(* Schneider Machine Expert - Basic project MEB, file version 2.7.0.0 *)
(* ProjectInformations: Name=Novo projeto *)

HARDWARE
  Cpu 0: TM221CE24R
  EthernetConfiguration: NetworkName=M221, IpAllocationMode=FixedAddress, IpAddress=0.0.0.0, SubnetMask=0.0.0.0
  SerialLineConfiguration: Baud=Baud19200, Parity=ParityEven, DataBits=DataBits8, StopBits=StopBits1, PhysicalMedium=PhysicalMediumRs485, TransmissionMode=TransmissionModeModbusRtu, SlaveId=1, Addressing=SlaveAddressing
  MastTask: UsePeriodScanMode=false, PeriodScan=100
  FastTask: Period=255
  CpuBehavior: StartingMode=StartAsPreviousState, AutoSaveRamOnEeprom=true, WatchdogPeriod=250

SYMBOLS  (address, symbol, comment, settings)
  %M0       AUX_PAI_EMER
  %M1       AUX_PAI_LOCA
  %M2       AUX_PAI_REMO
  %M3       CMD_PAI_MOT1_LIGA
  %M4       CMD_PAI_MOT1_DESL
  %M5       CMD_PAI_MOT2_LIGA
  %M6       CMD_PAI_MOT2_DESL
  %M50      HAB_MOT1
  %M51      HAB_MOT2
  %M100     CMD_IHM_INICIO
  %M101     CMD_IHM_FIM
  %I0.0     PAI_EMER
  %I0.1     PAI_LOCA
  %I0.2     PAI_REMO
  %I0.3     PAI_MOT1_LIGA
  %I0.4     PAI_MOT1_DESL
  %I0.5     PAI_MOT2_LIG
  %I0.6     PAI_MOT2_DESL
  %Q0.1     MOT1
  %Q0.2     MOT2

POU Novo POU
  (* SectionNumber=0 *)

// Rung 0
  LD
